% RSLogix 500 project BLUEBANNER_BINWASHER_NOV_2_2021_BAK013.RSS, saved by version 11.00.00.00 %
PROJECT "JBT BIN"    % processor: MicroLogix 1200 %

PROGRAM FILES
  LAD 2   8 rungs
  LAD 3   3 rungs
  LAD 4   11 rungs
  LAD 5   28 rungs
  LAD 6   7 rungs
  LAD 7   17 rungs
  LAD 8   6 rungs
  LAD 9   27 rungs

DATA FILES
  O0 OUTPUT  4 elements
  I1 INPUT  4 elements
  S2 STATUS  66 elements
  B3 BINARY  3 elements
  T4 TIMER  19 elements
  C5 COUNTER  1 elements
  R6 CONTROL  1 elements
  N7 INTEGER  6 elements
  F8 FLOAT  1 elements
  L9   1 elements
  L10   2 elements

LADDER 2
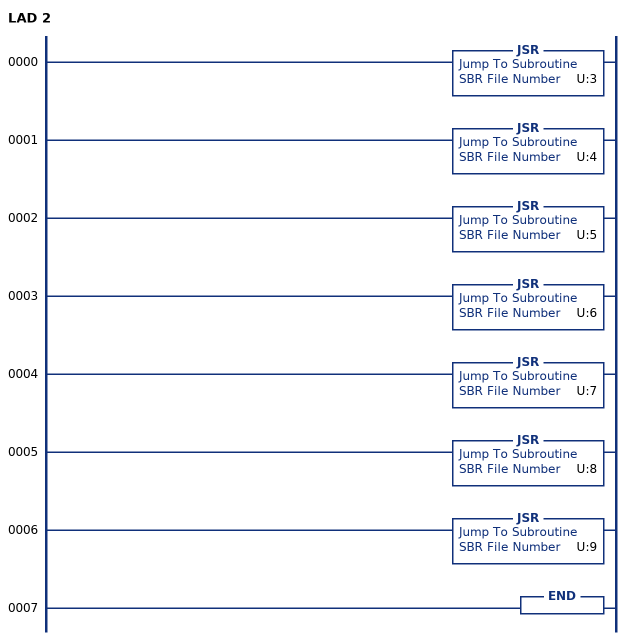
% Rung: 0 %
SOR JSR U:3 EOR
% Rung: 1 %
SOR JSR U:4 EOR
% Rung: 2 %
SOR JSR U:5 EOR
% Rung: 3 %
SOR JSR U:6 EOR
% Rung: 4 %
SOR JSR U:7 EOR
% Rung: 5 %
SOR JSR U:8 EOR
% Rung: 6 %
SOR JSR U:9 EOR
% Rung: 7 %
SOR END EOR

LADDER 3
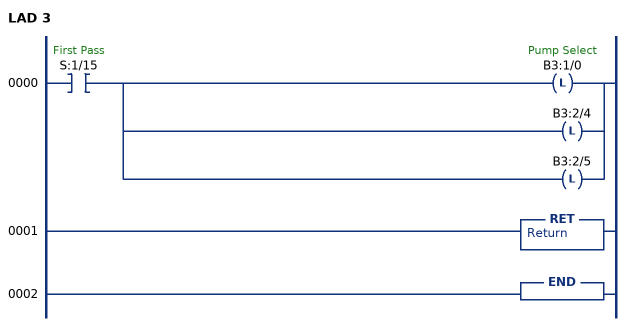
% Rung: 0 %
SOR XIC S:1/15 BST OTL B3:1/0 NXB BST OTL B3:2/4 NXB OTL B3:2/5 BND BND EOR
%   S:1/15  "First Pass" %
%   B3:1/0  "Pump Select" %
% Rung: 1 %
SOR RET EOR
% Rung: 2 %
SOR END EOR

LADDER 4
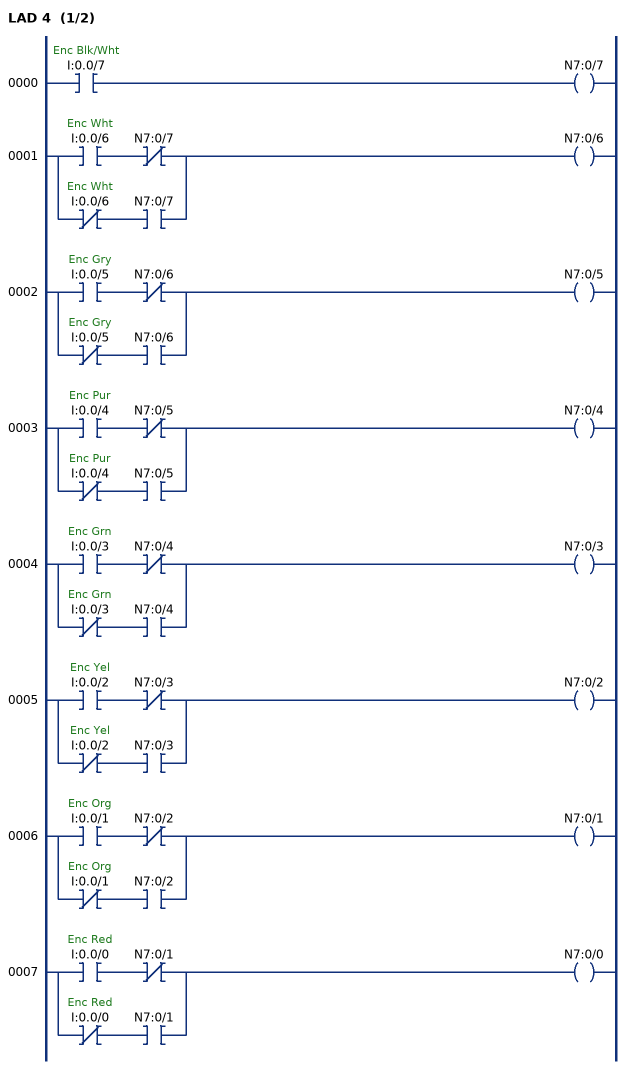
% Rung: 0 %
SOR XIC I:0.0/7 OTE N7:0/7 EOR
%   I:0.0/7  "Enc Blk/Wht" %
% Rung: 1 %
SOR BST XIC I:0.0/6 XIO N7:0/7 NXB XIO I:0.0/6 XIC N7:0/7 BND OTE N7:0/6 EOR
%   I:0.0/6  "Enc Wht" %
% Rung: 2 %
SOR BST XIC I:0.0/5 XIO N7:0/6 NXB XIO I:0.0/5 XIC N7:0/6 BND OTE N7:0/5 EOR
%   I:0.0/5  "Enc Gry" %
% Rung: 3 %
SOR BST XIC I:0.0/4 XIO N7:0/5 NXB XIO I:0.0/4 XIC N7:0/5 BND OTE N7:0/4 EOR
%   I:0.0/4  "Enc Pur" %
% Rung: 4 %
SOR BST XIC I:0.0/3 XIO N7:0/4 NXB XIO I:0.0/3 XIC N7:0/4 BND OTE N7:0/3 EOR
%   I:0.0/3  "Enc Grn" %
% Rung: 5 %
SOR BST XIC I:0.0/2 XIO N7:0/3 NXB XIO I:0.0/2 XIC N7:0/3 BND OTE N7:0/2 EOR
%   I:0.0/2  "Enc Yel" %
% Rung: 6 %
SOR BST XIC I:0.0/1 XIO N7:0/2 NXB XIO I:0.0/1 XIC N7:0/2 BND OTE N7:0/1 EOR
%   I:0.0/1  "Enc Org" %
% Rung: 7 %
SOR BST XIC I:0.0/0 XIO N7:0/1 NXB XIO I:0.0/0 XIC N7:0/1 BND OTE N7:0/0 EOR
%   I:0.0/0  "Enc Red" %

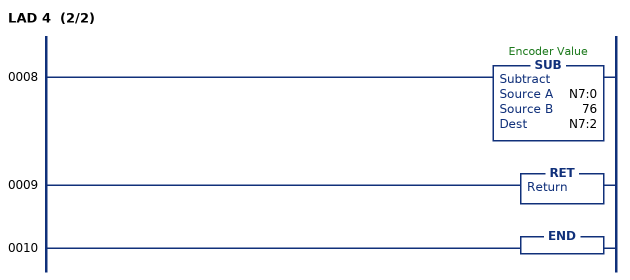
% Rung: 8 %
SOR SUB N7:0 76 N7:2 EOR
%   N7:2  "Encoder Value" %
% Rung: 9 %
SOR RET EOR
% Rung: 10 %
SOR END EOR

LADDER 5
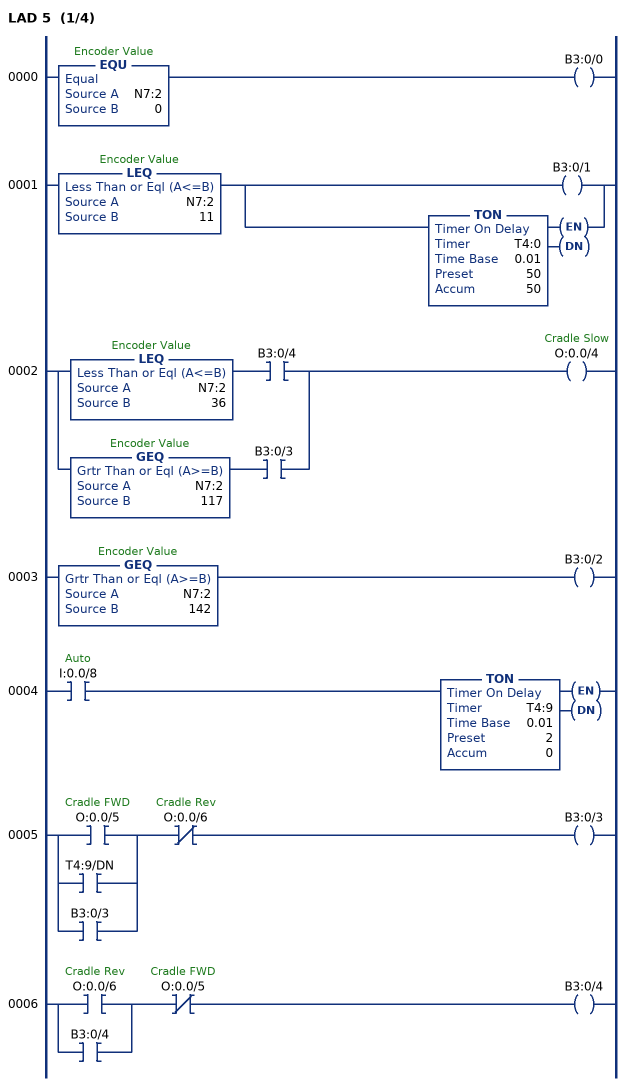
% Rung: 0 %
SOR EQU N7:2 0 OTE B3:0/0 EOR
%   N7:2  "Encoder Value" %
% Rung: 1 %
SOR LEQ N7:2 11 BST OTE B3:0/1 NXB TON T4:0 0.01 50 50 BND EOR
%   N7:2  "Encoder Value" %
% Rung: 2 %
SOR BST LEQ N7:2 36 XIC B3:0/4 NXB GEQ N7:2 117 XIC B3:0/3 BND OTE O:0.0/4 EOR
%   N7:2  "Encoder Value" %
%   O:0.0/4  "Cradle Slow" %
% Rung: 3 %
SOR GEQ N7:2 142 OTE B3:0/2 EOR
%   N7:2  "Encoder Value" %
% Rung: 4 %
SOR XIC I:0.0/8 TON T4:9 0.01 2 0 EOR
%   I:0.0/8  "Auto" %
% Rung: 5 %
SOR BST XIC O:0.0/5 NXB XIC T4:9/DN NXB XIC B3:0/3 BND XIO O:0.0/6 OTE B3:0/3 EOR
%   O:0.0/5  "Cradle FWD" %
%   O:0.0/6  "Cradle Rev" %
% Rung: 6 %
SOR BST XIC O:0.0/6 NXB XIC B3:0/4 BND XIO O:0.0/5 OTE B3:0/4 EOR
%   O:0.0/6  "Cradle Rev" %
%   O:0.0/5  "Cradle FWD" %

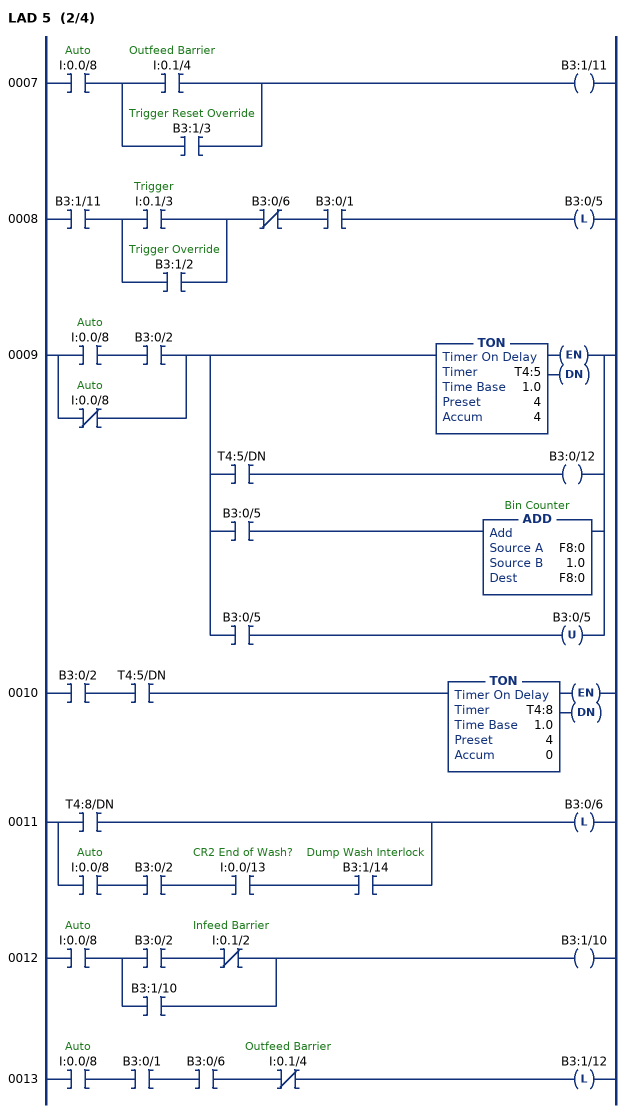
% Rung: 7 %
SOR XIC I:0.0/8 BST XIC I:0.1/4 NXB XIC B3:1/3 BND OTE B3:1/11 EOR
%   I:0.0/8  "Auto" %
%   I:0.1/4  "Outfeed Barrier" %
%   B3:1/3  "Trigger Reset Override" %
% Rung: 8 %
SOR XIC B3:1/11 BST XIC I:0.1/3 NXB XIC B3:1/2 BND XIO B3:0/6 XIC B3:0/1 OTL B3:0/5 EOR
%   I:0.1/3  "Trigger" %
%   B3:1/2  "Trigger Override" %
% Rung: 9 %
SOR BST XIC I:0.0/8 XIC B3:0/2 NXB XIO I:0.0/8 BND BST TON T4:5 1.0 4 4 NXB XIC T4:5/DN OTE B3:0/12 NXB BST XIC B3:0/5 ADD F8:0 1.0 F8:0 NXB XIC B3:0/5 OTU B3:0/5 BND BND EOR
%   I:0.0/8  "Auto" %
%   F8:0  "Bin Counter" %
% Rung: 10 %
SOR XIC B3:0/2 XIC T4:5/DN TON T4:8 1.0 4 0 EOR
% Rung: 11 %
SOR BST XIC T4:8/DN NXB XIC I:0.0/8 XIC B3:0/2 XIC I:0.0/13 XIC B3:1/14 BND OTL B3:0/6 EOR
%   I:0.0/8  "Auto" %
%   I:0.0/13  "CR2 End of Wash?" %
%   B3:1/14  "Dump Wash Interlock" %
% Rung: 12 %
SOR XIC I:0.0/8 BST XIC B3:0/2 XIO I:0.1/2 NXB XIC B3:1/10 BND OTE B3:1/10 EOR
%   I:0.0/8  "Auto" %
%   I:0.1/2  "Infeed Barrier" %
% Rung: 13 %
SOR XIC I:0.0/8 XIC B3:0/1 XIC B3:0/6 XIO I:0.1/4 OTL B3:1/12 EOR
%   I:0.0/8  "Auto" %
%   I:0.1/4  "Outfeed Barrier" %

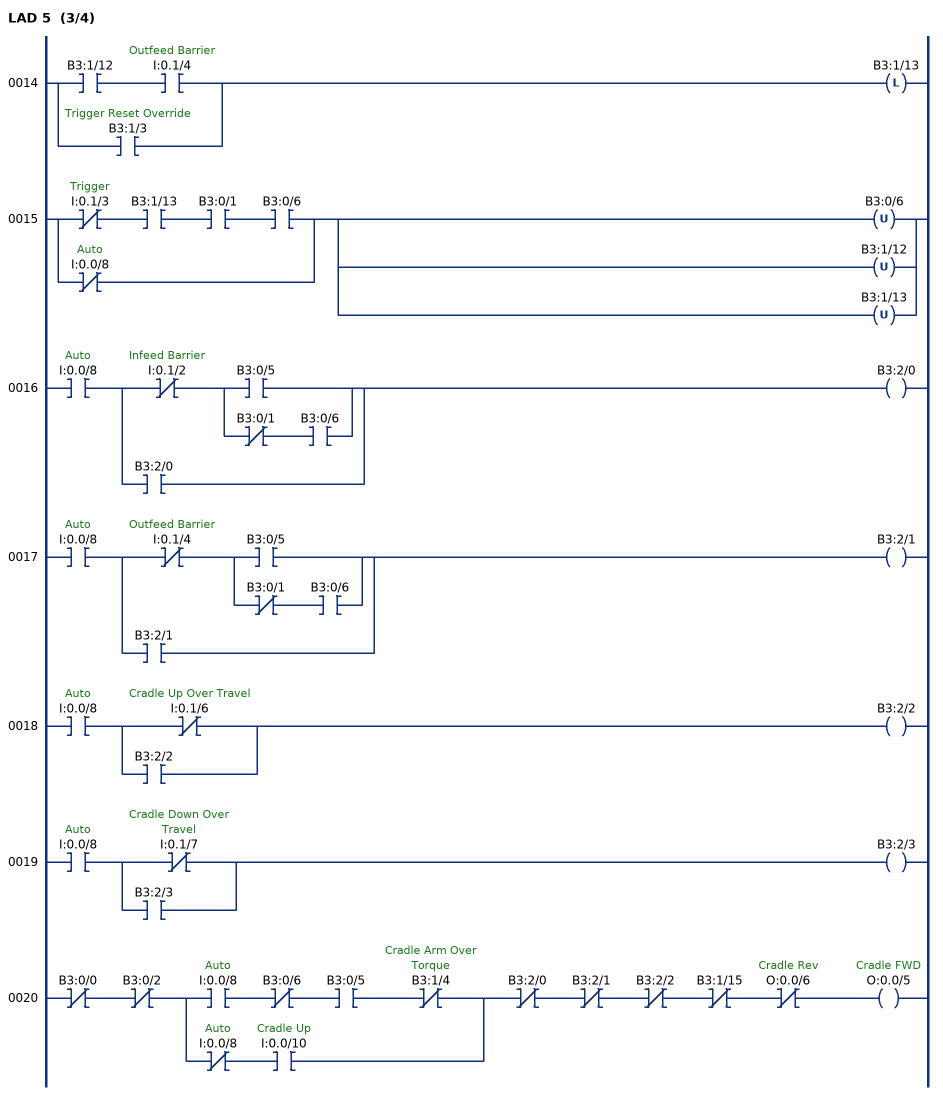
% Rung: 14 %
SOR BST XIC B3:1/12 XIC I:0.1/4 NXB XIC B3:1/3 BND OTL B3:1/13 EOR
%   I:0.1/4  "Outfeed Barrier" %
%   B3:1/3  "Trigger Reset Override" %
% Rung: 15 %
SOR BST XIO I:0.1/3 XIC B3:1/13 XIC B3:0/1 XIC B3:0/6 NXB XIO I:0.0/8 BND BST OTU B3:0/6 NXB BST OTU B3:1/12 NXB OTU B3:1/13 BND BND EOR
%   I:0.1/3  "Trigger" %
%   I:0.0/8  "Auto" %
% Rung: 16 %
SOR XIC I:0.0/8 BST XIO I:0.1/2 BST XIC B3:0/5 NXB XIO B3:0/1 XIC B3:0/6 BND NXB XIC B3:2/0 BND OTE B3:2/0 EOR
%   I:0.0/8  "Auto" %
%   I:0.1/2  "Infeed Barrier" %
% Rung: 17 %
SOR XIC I:0.0/8 BST XIO I:0.1/4 BST XIC B3:0/5 NXB XIO B3:0/1 XIC B3:0/6 BND NXB XIC B3:2/1 BND OTE B3:2/1 EOR
%   I:0.0/8  "Auto" %
%   I:0.1/4  "Outfeed Barrier" %
% Rung: 18 %
SOR XIC I:0.0/8 BST XIO I:0.1/6 NXB XIC B3:2/2 BND OTE B3:2/2 EOR
%   I:0.0/8  "Auto" %
%   I:0.1/6  "Cradle Up Over Travel" %
% Rung: 19 %
SOR XIC I:0.0/8 BST XIO I:0.1/7 NXB XIC B3:2/3 BND OTE B3:2/3 EOR
%   I:0.0/8  "Auto" %
%   I:0.1/7  "Cradle Down Over Travel" %
% Rung: 20 %
SOR XIO B3:0/0 XIO B3:0/2 BST XIC I:0.0/8 XIO B3:0/6 XIC B3:0/5 XIO B3:1/4 NXB XIO I:0.0/8 XIC I:0.0/10 BND XIO B3:2/0 XIO B3:2/1 XIO B3:2/2 XIO B3:1/15 XIO O:0.0/6 OTE O:0.0/5 EOR
%   I:0.0/8  "Auto" %
%   B3:1/4  "Cradle Arm Over Torque" %
%   I:0.0/10  "Cradle Up" %
%   O:0.0/6  "Cradle Rev" %
%   O:0.0/5  "Cradle FWD" %

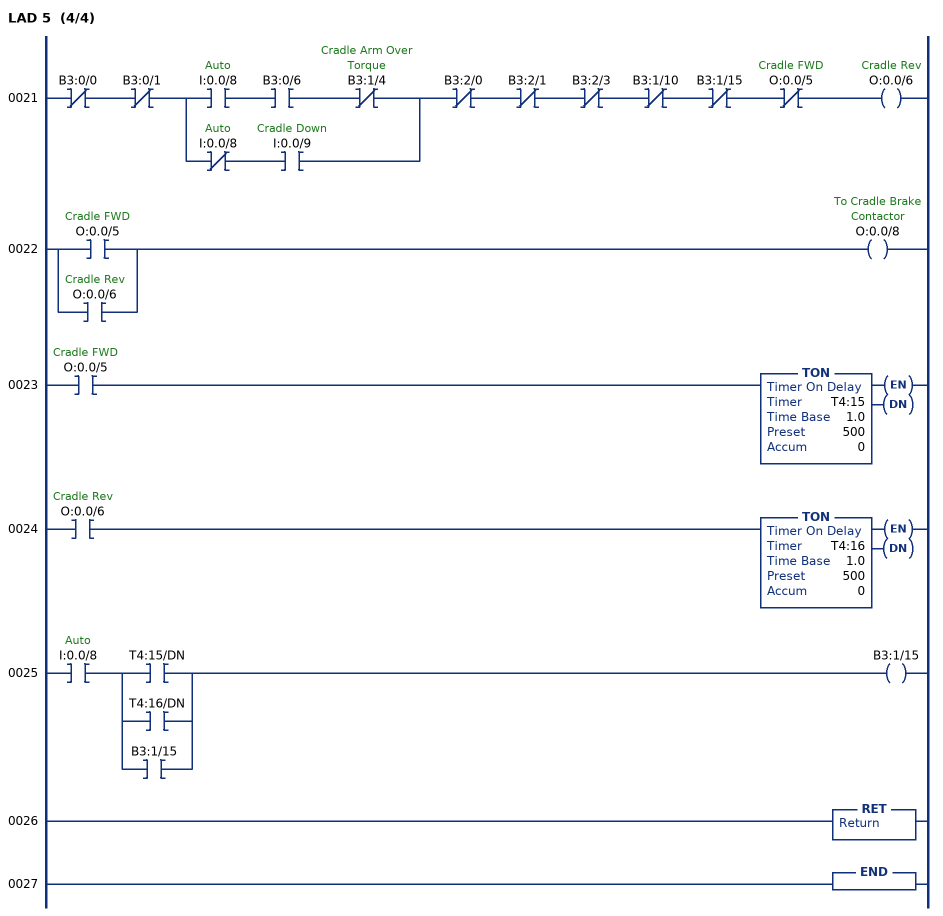
% Rung: 21 %
SOR XIO B3:0/0 XIO B3:0/1 BST XIC I:0.0/8 XIC B3:0/6 XIO B3:1/4 NXB XIO I:0.0/8 XIC I:0.0/9 BND XIO B3:2/0 XIO B3:2/1 XIO B3:2/3 XIO B3:1/10 XIO B3:1/15 XIO O:0.0/5 OTE O:0.0/6 EOR
%   I:0.0/8  "Auto" %
%   B3:1/4  "Cradle Arm Over Torque" %
%   I:0.0/9  "Cradle Down" %
%   O:0.0/5  "Cradle FWD" %
%   O:0.0/6  "Cradle Rev" %
% Rung: 22 %
SOR BST XIC O:0.0/5 NXB XIC O:0.0/6 BND OTE O:0.0/8 EOR
%   O:0.0/5  "Cradle FWD" %
%   O:0.0/6  "Cradle Rev" %
%   O:0.0/8  "To Cradle Brake Contactor" %
% Rung: 23 %
SOR XIC O:0.0/5 TON T4:15 1.0 500 0 EOR
%   O:0.0/5  "Cradle FWD" %
% Rung: 24 %
SOR XIC O:0.0/6 TON T4:16 1.0 500 0 EOR
%   O:0.0/6  "Cradle Rev" %
% Rung: 25 %
SOR XIC I:0.0/8 BST BST XIC T4:15/DN NXB XIC T4:16/DN BND NXB XIC B3:1/15 BND OTE B3:1/15 EOR
%   I:0.0/8  "Auto" %
% Rung: 26 %
SOR RET EOR
% Rung: 27 %
SOR END EOR

LADDER 6
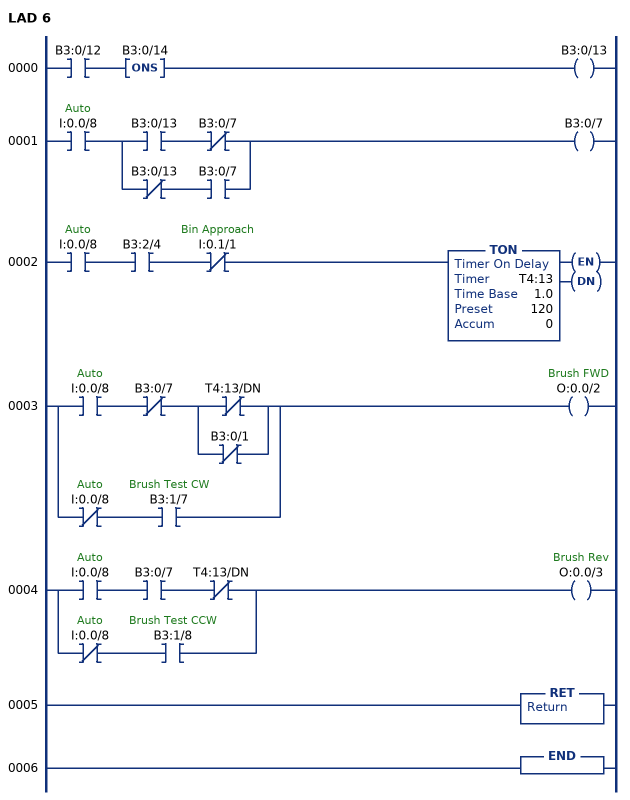
% Rung: 0 %
SOR XIC B3:0/12 ONS B3:0/14 OTE B3:0/13 EOR
% Rung: 1 %
SOR XIC I:0.0/8 BST XIC B3:0/13 XIO B3:0/7 NXB XIO B3:0/13 XIC B3:0/7 BND OTE B3:0/7 EOR
%   I:0.0/8  "Auto" %
% Rung: 2 %
SOR XIC I:0.0/8 XIC B3:2/4 XIO I:0.1/1 TON T4:13 1.0 120 0 EOR
%   I:0.0/8  "Auto" %
%   I:0.1/1  "Bin Approach" %
% Rung: 3 %
SOR BST XIC I:0.0/8 XIO B3:0/7 BST XIO T4:13/DN NXB XIO B3:0/1 BND NXB XIO I:0.0/8 XIC B3:1/7 BND OTE O:0.0/2 EOR
%   I:0.0/8  "Auto" %
%   B3:1/7  "Brush Test CW" %
%   O:0.0/2  "Brush FWD" %
% Rung: 4 %
SOR BST XIC I:0.0/8 XIC B3:0/7 XIO T4:13/DN NXB XIO I:0.0/8 XIC B3:1/8 BND OTE O:0.0/3 EOR
%   I:0.0/8  "Auto" %
%   B3:1/8  "Brush Test CCW" %
%   O:0.0/3  "Brush Rev" %
% Rung: 5 %
SOR RET EOR
% Rung: 6 %
SOR END EOR

LADDER 7
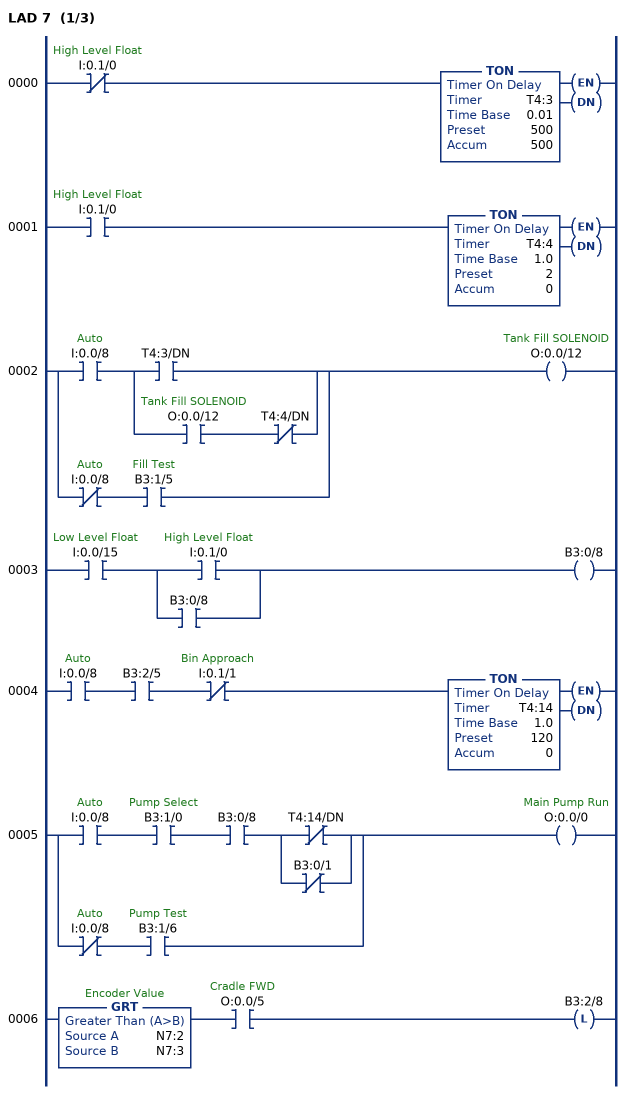
% Rung: 0 %
SOR XIO I:0.1/0 TON T4:3 0.01 500 500 EOR
%   I:0.1/0  "High Level Float" %
% Rung: 1 %
SOR XIC I:0.1/0 TON T4:4 1.0 2 0 EOR
%   I:0.1/0  "High Level Float" %
% Rung: 2 %
SOR BST XIC I:0.0/8 BST XIC T4:3/DN NXB XIC O:0.0/12 XIO T4:4/DN BND NXB XIO I:0.0/8 XIC B3:1/5 BND OTE O:0.0/12 EOR
%   I:0.0/8  "Auto" %
%   O:0.0/12  "Tank Fill SOLENOID" %
%   B3:1/5  "Fill Test" %
% Rung: 3 %
SOR XIC I:0.0/15 BST XIC I:0.1/0 NXB XIC B3:0/8 BND OTE B3:0/8 EOR
%   I:0.0/15  "Low Level Float" %
%   I:0.1/0  "High Level Float" %
% Rung: 4 %
SOR XIC I:0.0/8 XIC B3:2/5 XIO I:0.1/1 TON T4:14 1.0 120 0 EOR
%   I:0.0/8  "Auto" %
%   I:0.1/1  "Bin Approach" %
% Rung: 5 %
SOR BST XIC I:0.0/8 XIC B3:1/0 XIC B3:0/8 BST XIO T4:14/DN NXB XIO B3:0/1 BND NXB XIO I:0.0/8 XIC B3:1/6 BND OTE O:0.0/0 EOR
%   I:0.0/8  "Auto" %
%   B3:1/0  "Pump Select" %
%   B3:1/6  "Pump Test" %
%   O:0.0/0  "Main Pump Run" %
% Rung: 6 %
SOR GRT N7:2 N7:3 XIC O:0.0/5 OTL B3:2/8 EOR
%   N7:2  "Encoder Value" %
%   O:0.0/5  "Cradle FWD" %

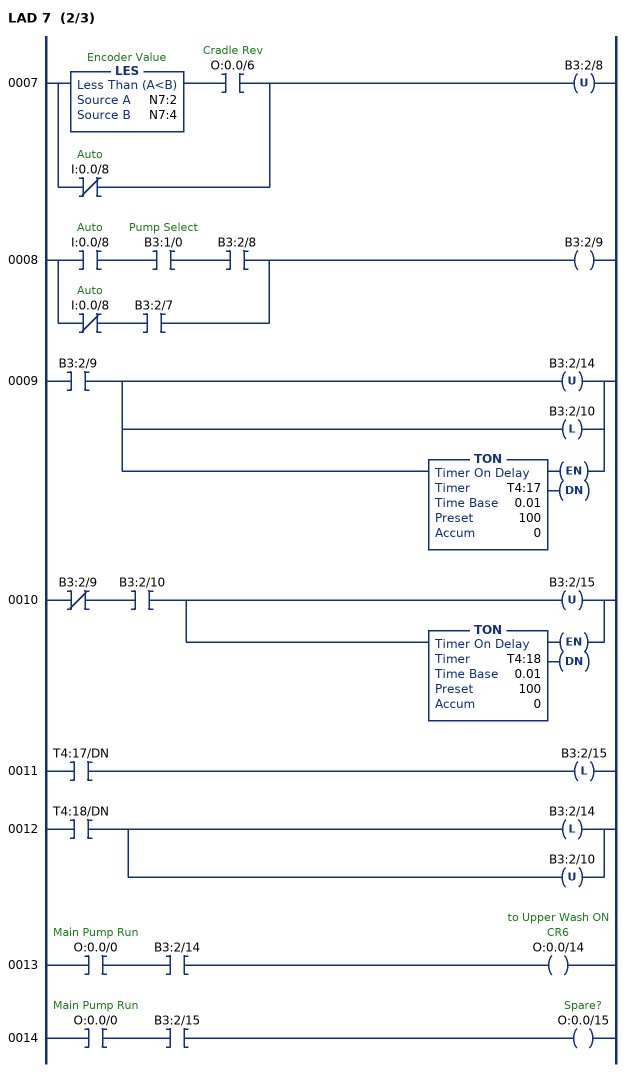
% Rung: 7 %
SOR BST LES N7:2 N7:4 XIC O:0.0/6 NXB XIO I:0.0/8 BND OTU B3:2/8 EOR
%   N7:2  "Encoder Value" %
%   O:0.0/6  "Cradle Rev" %
%   I:0.0/8  "Auto" %
% Rung: 8 %
SOR BST XIC I:0.0/8 XIC B3:1/0 XIC B3:2/8 NXB XIO I:0.0/8 XIC B3:2/7 BND OTE B3:2/9 EOR
%   I:0.0/8  "Auto" %
%   B3:1/0  "Pump Select" %
% Rung: 9 %
SOR XIC B3:2/9 BST OTU B3:2/14 NXB BST OTL B3:2/10 NXB TON T4:17 0.01 100 0 BND BND EOR
% Rung: 10 %
SOR XIO B3:2/9 XIC B3:2/10 BST OTU B3:2/15 NXB TON T4:18 0.01 100 0 BND EOR
% Rung: 11 %
SOR XIC T4:17/DN OTL B3:2/15 EOR
% Rung: 12 %
SOR XIC T4:18/DN BST OTL B3:2/14 NXB OTU B3:2/10 BND EOR
% Rung: 13 %
SOR XIC O:0.0/0 XIC B3:2/14 OTE O:0.0/14 EOR
%   O:0.0/0  "Main Pump Run" %
%   O:0.0/14  "to Upper Wash ON CR6" %
% Rung: 14 %
SOR XIC O:0.0/0 XIC B3:2/15 OTE O:0.0/15 EOR
%   O:0.0/0  "Main Pump Run" %
%   O:0.0/15  "Spare?" %

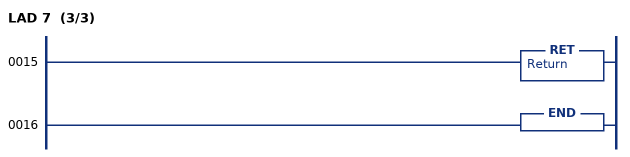
% Rung: 15 %
SOR RET EOR
% Rung: 16 %
SOR END EOR

LADDER 8
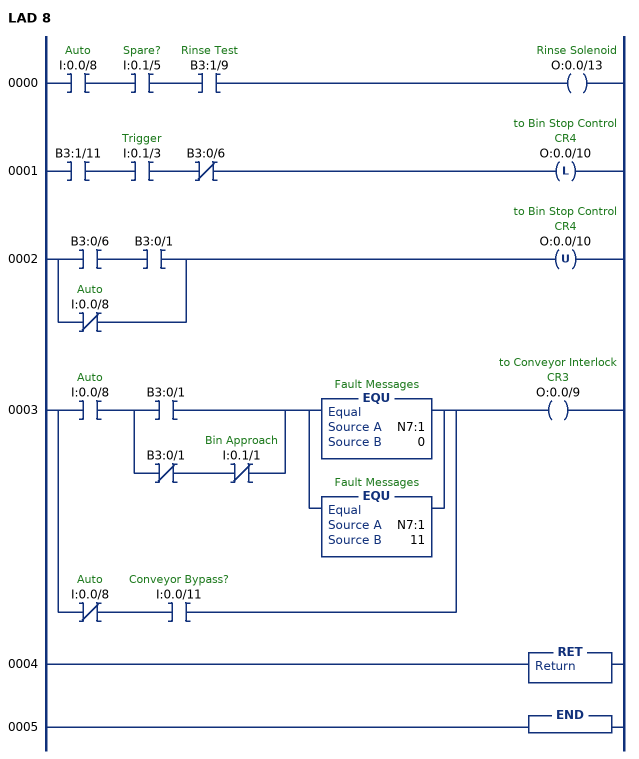
% Rung: 0 %
SOR XIC I:0.0/8 XIC I:0.1/5 XIC B3:1/9 OTE O:0.0/13 EOR
%   I:0.0/8  "Auto" %
%   I:0.1/5  "Spare?" %
%   B3:1/9  "Rinse Test" %
%   O:0.0/13  "Rinse Solenoid" %
% Rung: 1 %
SOR XIC B3:1/11 XIC I:0.1/3 XIO B3:0/6 OTL O:0.0/10 EOR
%   I:0.1/3  "Trigger" %
%   O:0.0/10  "to Bin Stop Control CR4" %
% Rung: 2 %
SOR BST XIC B3:0/6 XIC B3:0/1 NXB XIO I:0.0/8 BND OTU O:0.0/10 EOR
%   I:0.0/8  "Auto" %
%   O:0.0/10  "to Bin Stop Control CR4" %
% Rung: 3 %
SOR BST XIC I:0.0/8 BST XIC B3:0/1 NXB XIO B3:0/1 XIO I:0.1/1 BND BST EQU N7:1 0 NXB EQU N7:1 11 BND NXB XIO I:0.0/8 XIC I:0.0/11 BND OTE O:0.0/9 EOR
%   I:0.0/8  "Auto" %
%   I:0.1/1  "Bin Approach" %
%   N7:1  "Fault Messages" %
%   I:0.0/11  "Conveyor Bypass?" %
%   O:0.0/9  "to Conveyor Interlock CR3" %
% Rung: 4 %
SOR RET EOR
% Rung: 5 %
SOR END EOR

LADDER 9
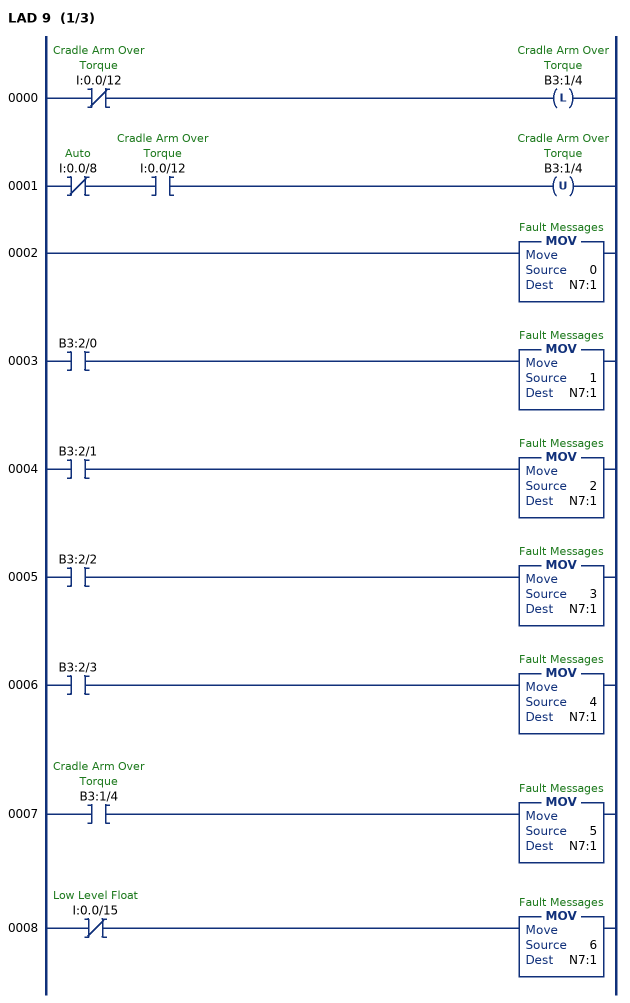
% Rung: 0 %
SOR XIO I:0.0/12 OTL B3:1/4 EOR
%   I:0.0/12  "Cradle Arm Over Torque" %
%   B3:1/4  "Cradle Arm Over Torque" %
% Rung: 1 %
SOR XIO I:0.0/8 XIC I:0.0/12 OTU B3:1/4 EOR
%   I:0.0/8  "Auto" %
%   I:0.0/12  "Cradle Arm Over Torque" %
%   B3:1/4  "Cradle Arm Over Torque" %
% Rung: 2 %
SOR MOV 0 N7:1 EOR
%   N7:1  "Fault Messages" %
% Rung: 3 %
SOR XIC B3:2/0 MOV 1 N7:1 EOR
%   N7:1  "Fault Messages" %
% Rung: 4 %
SOR XIC B3:2/1 MOV 2 N7:1 EOR
%   N7:1  "Fault Messages" %
% Rung: 5 %
SOR XIC B3:2/2 MOV 3 N7:1 EOR
%   N7:1  "Fault Messages" %
% Rung: 6 %
SOR XIC B3:2/3 MOV 4 N7:1 EOR
%   N7:1  "Fault Messages" %
% Rung: 7 %
SOR XIC B3:1/4 MOV 5 N7:1 EOR
%   B3:1/4  "Cradle Arm Over Torque" %
%   N7:1  "Fault Messages" %
% Rung: 8 %
SOR XIO I:0.0/15 MOV 6 N7:1 EOR
%   I:0.0/15  "Low Level Float" %
%   N7:1  "Fault Messages" %

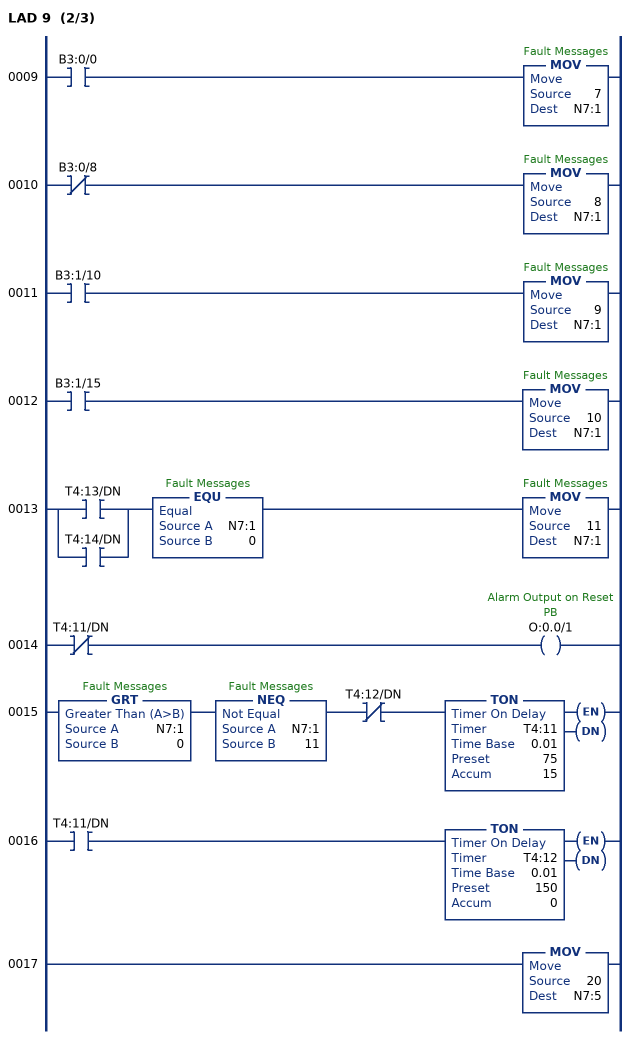
% Rung: 9 %
SOR XIC B3:0/0 MOV 7 N7:1 EOR
%   N7:1  "Fault Messages" %
% Rung: 10 %
SOR XIO B3:0/8 MOV 8 N7:1 EOR
%   N7:1  "Fault Messages" %
% Rung: 11 %
SOR XIC B3:1/10 MOV 9 N7:1 EOR
%   N7:1  "Fault Messages" %
% Rung: 12 %
SOR XIC B3:1/15 MOV 10 N7:1 EOR
%   N7:1  "Fault Messages" %
% Rung: 13 %
SOR BST XIC T4:13/DN NXB XIC T4:14/DN BND EQU N7:1 0 MOV 11 N7:1 EOR
%   N7:1  "Fault Messages" %
% Rung: 14 %
SOR XIO T4:11/DN OTE O:0.0/1 EOR
%   O:0.0/1  "Alarm Output on Reset PB" %
% Rung: 15 %
SOR GRT N7:1 0 NEQ N7:1 11 XIO T4:12/DN TON T4:11 0.01 75 15 EOR
%   N7:1  "Fault Messages" %
% Rung: 16 %
SOR XIC T4:11/DN TON T4:12 0.01 150 0 EOR
% Rung: 17 %
SOR MOV 20 N7:5 EOR

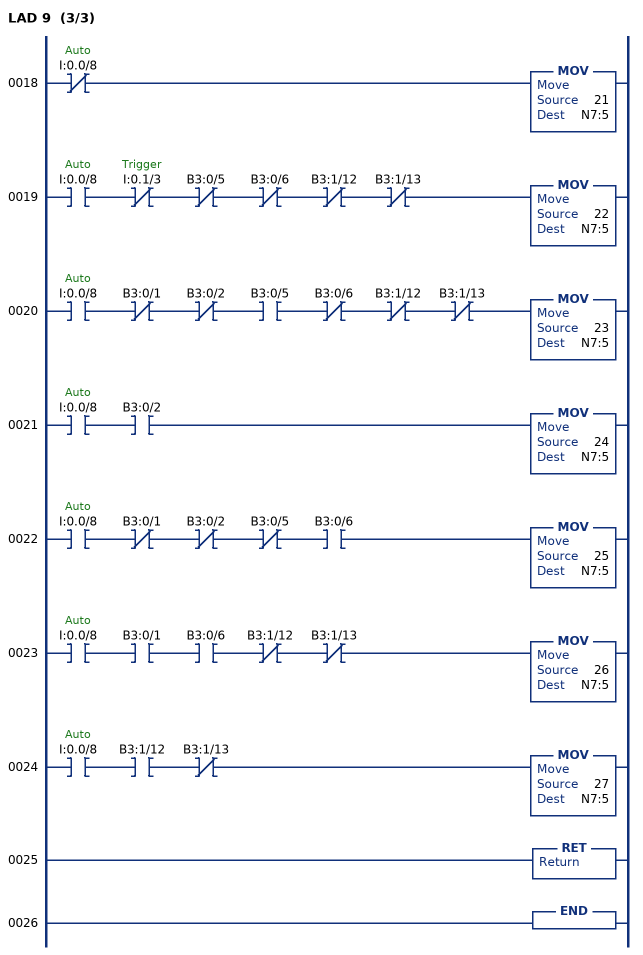
% Rung: 18 %
SOR XIO I:0.0/8 MOV 21 N7:5 EOR
%   I:0.0/8  "Auto" %
% Rung: 19 %
SOR XIC I:0.0/8 XIO I:0.1/3 XIO B3:0/5 XIO B3:0/6 XIO B3:1/12 XIO B3:1/13 MOV 22 N7:5 EOR
%   I:0.0/8  "Auto" %
%   I:0.1/3  "Trigger" %
% Rung: 20 %
SOR XIC I:0.0/8 XIO B3:0/1 XIO B3:0/2 XIC B3:0/5 XIO B3:0/6 XIO B3:1/12 XIO B3:1/13 MOV 23 N7:5 EOR
%   I:0.0/8  "Auto" %
% Rung: 21 %
SOR XIC I:0.0/8 XIC B3:0/2 MOV 24 N7:5 EOR
%   I:0.0/8  "Auto" %
% Rung: 22 %
SOR XIC I:0.0/8 XIO B3:0/1 XIO B3:0/2 XIO B3:0/5 XIC B3:0/6 MOV 25 N7:5 EOR
%   I:0.0/8  "Auto" %
% Rung: 23 %
SOR XIC I:0.0/8 XIC B3:0/1 XIC B3:0/6 XIO B3:1/12 XIO B3:1/13 MOV 26 N7:5 EOR
%   I:0.0/8  "Auto" %
% Rung: 24 %
SOR XIC I:0.0/8 XIC B3:1/12 XIO B3:1/13 MOV 27 N7:5 EOR
%   I:0.0/8  "Auto" %
% Rung: 25 %
SOR RET EOR
% Rung: 26 %
SOR END EOR

OTHER DOCUMENTED ADDRESSES
  I:0.0/14  "Optional Cradle Brake Aux"
  O:0.0/11  "Spare?"
  T4:5.PRE  "Clean CW"
  T4:8.PRE  "Clean CCW"

REVISION NOTES
  0: encoder edit for 9to11 is ok to go up

DATA TABLE (non-zero values as saved)
DATA B3
% B3:0 % 0X5C02 0X4223 0X4030
DATA T4
% .PRE .ACC %
% T4:0 % 50 50
% T4:1 % 1 0
% T4:2 % 1 0
% T4:3 % 500 500
% T4:4 % 2 0
% T4:5 % 4 4
% T4:6 % 658 0
% T4:7 % 375 500
% T4:8 % 4 0
% T4:9 % 2 0
% T4:10 % 500 0
% T4:11 % 75 15
% T4:12 % 150 0
% T4:13 % 120 0
% T4:14 % 120 0
% T4:15 % 500 0
% T4:16 % 500 0
% T4:17 % 100 0
% T4:18 % 100 0
DATA N7
% N7:0 % 86 8 10 65 130 21
DATA F8
% F8:0 % 23
